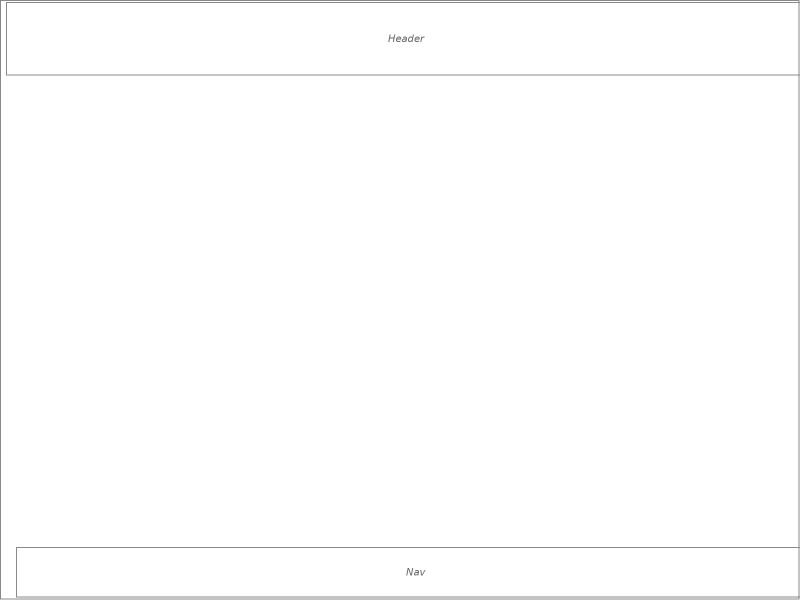
VISUALIZATION MainScreen  // 800x600
    Frame (6,2 800x73)
        shows Header()
    Frame (16,547 800x50)
        shows Nav()
END_VISUALIZATION

(* stored: Version 1.1.0.1, ProductVersion 3.1.4024.12
   Visu MainScreen: Id {73012c66-31f6-4eca-a54e-2f1314361f5a} *)
